% RSLogix 500 project LAB 5_BGJ.RSS, saved by version 8.40.00.08 %
PROJECT "MAN_MODE"    % processor: SLC 500, 1747-L541 %

PROGRAM FILES
  LAD 2   67 rungs

DATA FILES
  O0 OUTPUT  68 elements
  I1 INPUT  68 elements
  S2 STATUS  164 elements
  B3 BINARY  2 elements
  T4 TIMER  20 elements
  C5 COUNTER  2 elements
  R6 CONTROL  1 elements
  N7 INTEGER  1 elements
  F8 FLOAT  1 elements
  N10 PV_OUTPUTS  32 elements
  N11 PV_INPUTS  32 elements

LADDER 2
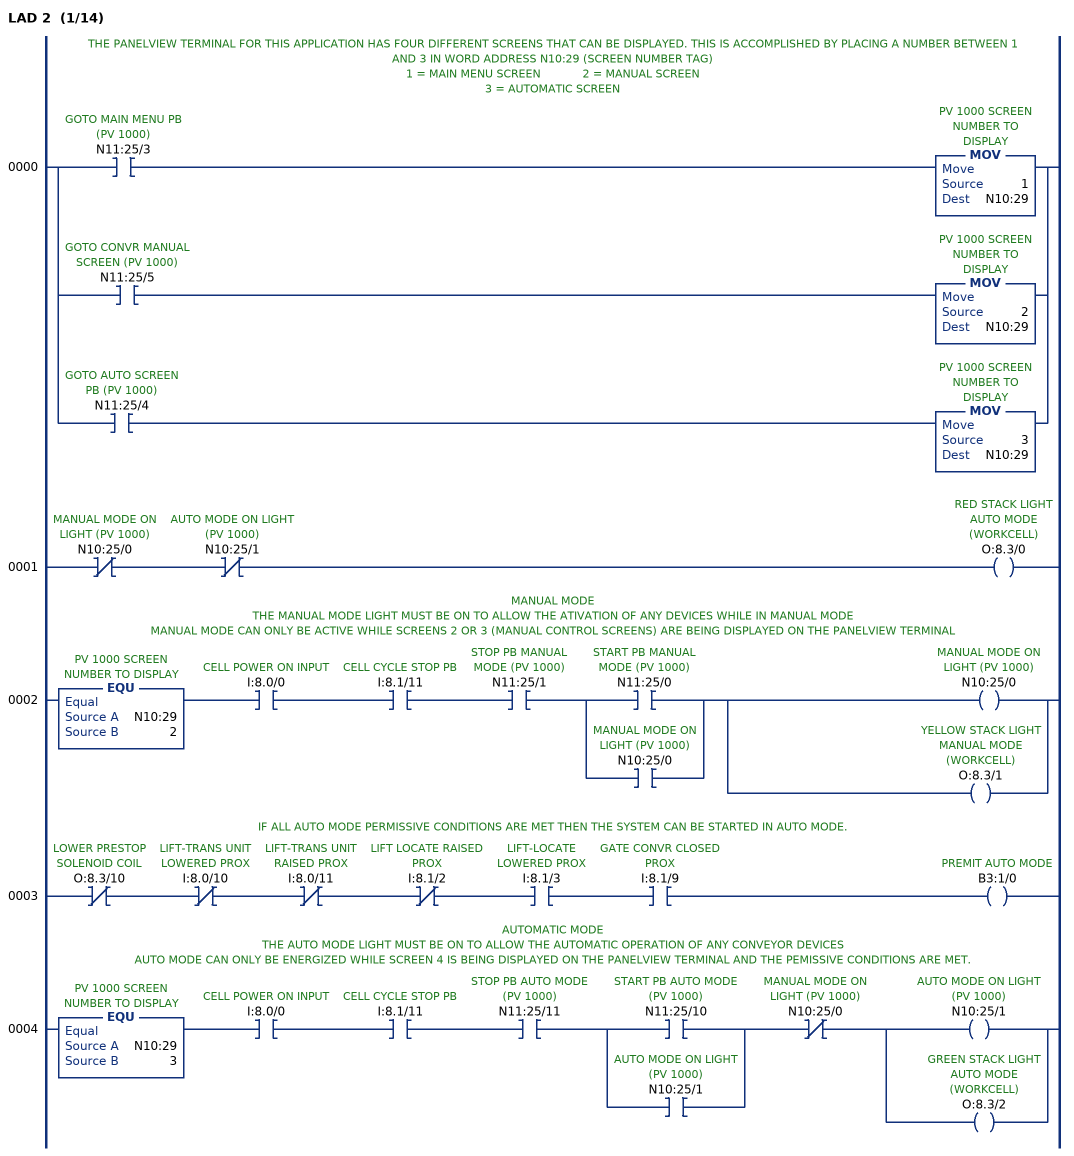
% Rung: 0 %
% THE PANELVIEW TERMINAL FOR THIS APPLICATION HAS FOUR DIFFERENT SCREENS THAT CAN BE DISPLAYED. THIS IS ACCOMPLISHED BY PLACING A NUMBER BETWEEN 1 AND 3 IN WORD ADDRESS N10:29 (SCREEN NUMBER TAG)
% 
% 1 = MAIN MENU SCREEN            2 = MANUAL SCREEN
% 3 = AUTOMATIC SCREEN %
SOR BST XIC N11:25/3 MOV 1 N10:29 NXB XIC N11:25/5 MOV 2 N10:29 NXB XIC N11:25/4 MOV 3 N10:29 BND EOR
%   N11:25/3  "GOTO MAIN MENU PB (PV 1000)" %
%   N10:29  "PV 1000 SCREEN NUMBER TO DISPLAY" %
%   N11:25/5  "GOTO CONVR MANUAL SCREEN (PV 1000)" %
%   N11:25/4  "GOTO AUTO SCREEN PB (PV 1000)" %
% Rung: 1 %
SOR XIO N10:25/0 XIO N10:25/1 OTE O:8.3/0 EOR
%   N10:25/0  "MANUAL MODE ON LIGHT (PV 1000)" %
%   N10:25/1  "AUTO MODE ON LIGHT (PV 1000)" %
%   O:8.3/0  "RED STACK LIGHT AUTO MODE (WORKCELL)" %
% Rung: 2 %
% MANUAL MODE
% 
% THE MANUAL MODE LIGHT MUST BE ON TO ALLOW THE ATIVATION OF ANY DEVICES WHILE IN MANUAL MODE
% MANUAL MODE CAN ONLY BE ACTIVE WHILE SCREENS 2 OR 3 (MANUAL CONTROL SCREENS) ARE BEING DISPLAYED ON THE PANELVIEW TERMINAL %
SOR EQU N10:29 2 XIC I:8.0/0 XIC I:8.1/11 XIC N11:25/1 BST XIC N11:25/0 NXB XIC N10:25/0 BND BST OTE N10:25/0 NXB OTE O:8.3/1 BND EOR
%   N10:29  "PV 1000 SCREEN NUMBER TO DISPLAY" %
%   I:8.0/0  "CELL POWER ON INPUT" %
%   I:8.1/11  "CELL CYCLE STOP PB" %
%   N11:25/1  "STOP PB MANUAL MODE (PV 1000)" %
%   N11:25/0  "START PB MANUAL MODE (PV 1000)" %
%   N10:25/0  "MANUAL MODE ON LIGHT (PV 1000)" %
%   O:8.3/1  "YELLOW STACK LIGHT MANUAL MODE (WORKCELL)" %
% Rung: 3 %
% IF ALL AUTO MODE PERMISSIVE CONDITIONS ARE MET THEN THE SYSTEM CAN BE STARTED IN AUTO MODE. %
SOR XIO O:8.3/10 XIO I:8.0/10 XIO I:8.0/11 XIO I:8.1/2 XIC I:8.1/3 XIC I:8.1/9 OTE B3:1/0 EOR
%   O:8.3/10  "LOWER PRESTOP SOLENOID COIL" %
%   I:8.0/10  "LIFT-TRANS UNIT LOWERED PROX" %
%   I:8.0/11  "LIFT-TRANS UNIT RAISED PROX" %
%   I:8.1/2  "LIFT LOCATE RAISED PROX" %
%   I:8.1/3  "LIFT-LOCATE LOWERED PROX" %
%   I:8.1/9  "GATE CONVR CLOSED PROX" %
%   B3:1/0  "PREMIT AUTO MODE" %
% Rung: 4 %
% AUTOMATIC MODE
% 
% THE AUTO MODE LIGHT MUST BE ON TO ALLOW THE AUTOMATIC OPERATION OF ANY CONVEYOR DEVICES
% 
% AUTO MODE CAN ONLY BE ENERGIZED WHILE SCREEN 4 IS BEING DISPLAYED ON THE PANELVIEW TERMINAL AND THE PEMISSIVE CONDITIONS ARE MET. %
SOR EQU N10:29 3 XIC I:8.0/0 XIC I:8.1/11 XIC N11:25/11 BST XIC N11:25/10 NXB XIC N10:25/1 BND XIO N10:25/0 BST OTE N10:25/1 NXB OTE O:8.3/2 BND EOR
%   N10:29  "PV 1000 SCREEN NUMBER TO DISPLAY" %
%   I:8.0/0  "CELL POWER ON INPUT" %
%   I:8.1/11  "CELL CYCLE STOP PB" %
%   N11:25/11  "STOP PB AUTO MODE (PV 1000)" %
%   N11:25/10  "START PB AUTO MODE (PV 1000)" %
%   N10:25/1  "AUTO MODE ON LIGHT (PV 1000)" %
%   N10:25/0  "MANUAL MODE ON LIGHT (PV 1000)" %
%   O:8.3/2  "GREEN STACK LIGHT AUTO MODE (WORKCELL)" %

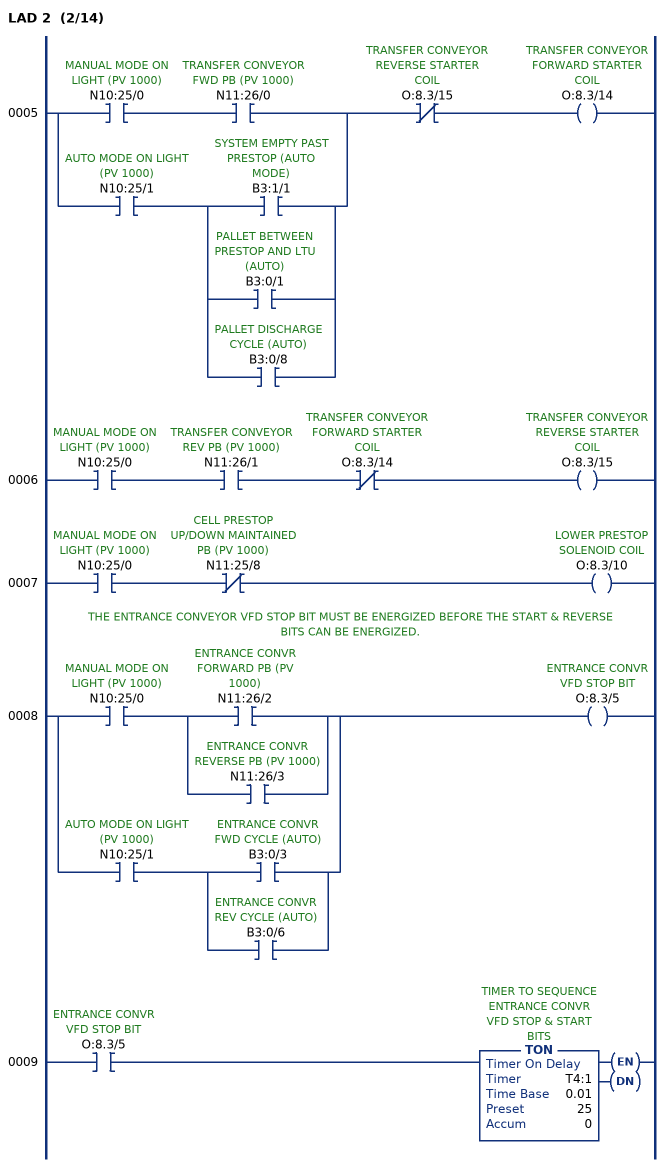
% Rung: 5 %
SOR BST XIC N10:25/0 XIC N11:26/0 NXB XIC N10:25/1 BST XIC B3:1/1 NXB XIC B3:0/1 NXB XIC B3:0/8 BND BND XIO O:8.3/15 OTE O:8.3/14 EOR
%   N10:25/0  "MANUAL MODE ON LIGHT (PV 1000)" %
%   N11:26/0  "TRANSFER CONVEYOR FWD PB (PV 1000)" %
%   N10:25/1  "AUTO MODE ON LIGHT (PV 1000)" %
%   B3:1/1  "SYSTEM EMPTY PAST PRESTOP (AUTO MODE)" %
%   B3:0/1  "PALLET BETWEEN PRESTOP AND LTU (AUTO)" %
%   B3:0/8  "PALLET DISCHARGE CYCLE (AUTO)" %
%   O:8.3/15  "TRANSFER CONVEYOR REVERSE STARTER COIL" %
%   O:8.3/14  "TRANSFER CONVEYOR FORWARD STARTER COIL" %
% Rung: 6 %
SOR XIC N10:25/0 XIC N11:26/1 XIO O:8.3/14 OTE O:8.3/15 EOR
%   N10:25/0  "MANUAL MODE ON LIGHT (PV 1000)" %
%   N11:26/1  "TRANSFER CONVEYOR REV PB (PV 1000)" %
%   O:8.3/14  "TRANSFER CONVEYOR FORWARD STARTER COIL" %
%   O:8.3/15  "TRANSFER CONVEYOR REVERSE STARTER COIL" %
% Rung: 7 %
SOR XIC N10:25/0 XIO N11:25/8 OTE O:8.3/10 EOR
%   N10:25/0  "MANUAL MODE ON LIGHT (PV 1000)" %
%   N11:25/8  "CELL PRESTOP UP/DOWN MAINTAINED PB (PV 1000)" %
%   O:8.3/10  "LOWER PRESTOP SOLENOID COIL" %
% Rung: 8 %
% THE ENTRANCE CONVEYOR VFD STOP BIT MUST BE ENERGIZED BEFORE THE START & REVERSE BITS CAN BE ENERGIZED. %
SOR BST XIC N10:25/0 BST XIC N11:26/2 NXB XIC N11:26/3 BND NXB XIC N10:25/1 BST XIC B3:0/3 NXB XIC B3:0/6 BND BND OTE O:8.3/5 EOR
%   N10:25/0  "MANUAL MODE ON LIGHT (PV 1000)" %
%   N11:26/2  "ENTRANCE CONVR FORWARD PB (PV 1000)" %
%   N11:26/3  "ENTRANCE CONVR REVERSE PB (PV 1000)" %
%   N10:25/1  "AUTO MODE ON LIGHT (PV 1000)" %
%   B3:0/3  "ENTRANCE CONVR FWD CYCLE (AUTO)" %
%   B3:0/6  "ENTRANCE CONVR REV CYCLE (AUTO)" %
%   O:8.3/5  "ENTRANCE CONVR VFD STOP BIT" %
% Rung: 9 %
SOR XIC O:8.3/5 TON T4:1 0.01 25 0 EOR
%   O:8.3/5  "ENTRANCE CONVR VFD STOP BIT" %
%   T4:1  "TIMER TO SEQUENCE ENTRANCE CONVR VFD STOP & START BITS" %

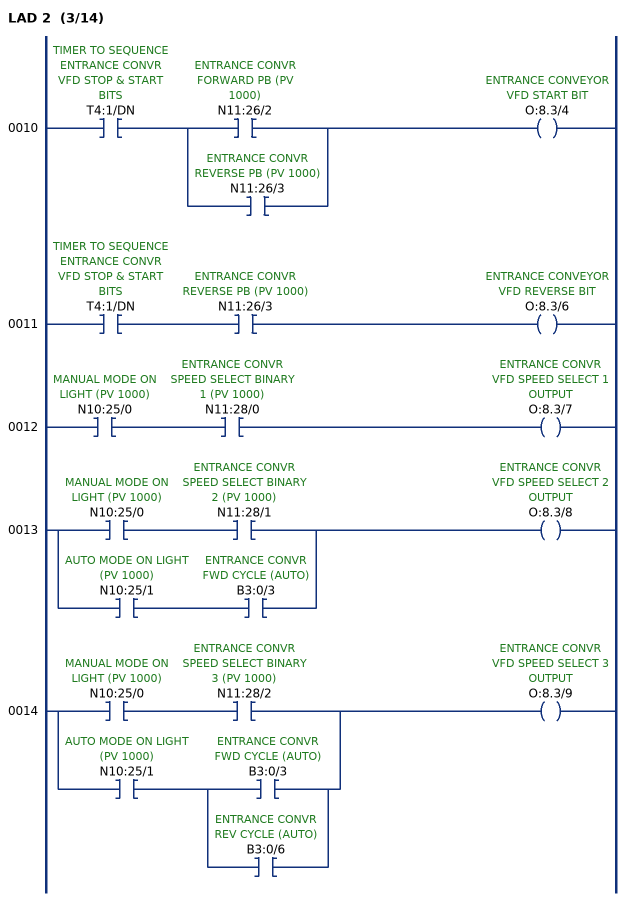
% Rung: 10 %
SOR XIC T4:1/DN BST XIC N11:26/2 NXB XIC N11:26/3 BND OTE O:8.3/4 EOR
%   T4:1  "TIMER TO SEQUENCE ENTRANCE CONVR VFD STOP & START BITS" %
%   N11:26/2  "ENTRANCE CONVR FORWARD PB (PV 1000)" %
%   N11:26/3  "ENTRANCE CONVR REVERSE PB (PV 1000)" %
%   O:8.3/4  "ENTRANCE CONVEYOR VFD START BIT" %
% Rung: 11 %
SOR XIC T4:1/DN XIC N11:26/3 OTE O:8.3/6 EOR
%   T4:1  "TIMER TO SEQUENCE ENTRANCE CONVR VFD STOP & START BITS" %
%   N11:26/3  "ENTRANCE CONVR REVERSE PB (PV 1000)" %
%   O:8.3/6  "ENTRANCE CONVEYOR VFD REVERSE BIT" %
% Rung: 12 %
SOR XIC N10:25/0 XIC N11:28/0 OTE O:8.3/7 EOR
%   N10:25/0  "MANUAL MODE ON LIGHT (PV 1000)" %
%   N11:28/0  "ENTRANCE CONVR SPEED SELECT BINARY 1 (PV 1000)" %
%   O:8.3/7  "ENTRANCE CONVR VFD SPEED SELECT 1 OUTPUT" %
% Rung: 13 %
SOR BST XIC N10:25/0 XIC N11:28/1 NXB XIC N10:25/1 XIC B3:0/3 BND OTE O:8.3/8 EOR
%   N10:25/0  "MANUAL MODE ON LIGHT (PV 1000)" %
%   N11:28/1  "ENTRANCE CONVR SPEED SELECT BINARY 2 (PV 1000)" %
%   N10:25/1  "AUTO MODE ON LIGHT (PV 1000)" %
%   B3:0/3  "ENTRANCE CONVR FWD CYCLE (AUTO)" %
%   O:8.3/8  "ENTRANCE CONVR VFD SPEED SELECT 2 OUTPUT" %
% Rung: 14 %
SOR BST XIC N10:25/0 XIC N11:28/2 NXB XIC N10:25/1 BST XIC B3:0/3 NXB XIC B3:0/6 BND BND OTE O:8.3/9 EOR
%   N10:25/0  "MANUAL MODE ON LIGHT (PV 1000)" %
%   N11:28/2  "ENTRANCE CONVR SPEED SELECT BINARY 3 (PV 1000)" %
%   N10:25/1  "AUTO MODE ON LIGHT (PV 1000)" %
%   B3:0/3  "ENTRANCE CONVR FWD CYCLE (AUTO)" %
%   B3:0/6  "ENTRANCE CONVR REV CYCLE (AUTO)" %
%   O:8.3/9  "ENTRANCE CONVR VFD SPEED SELECT 3 OUTPUT" %

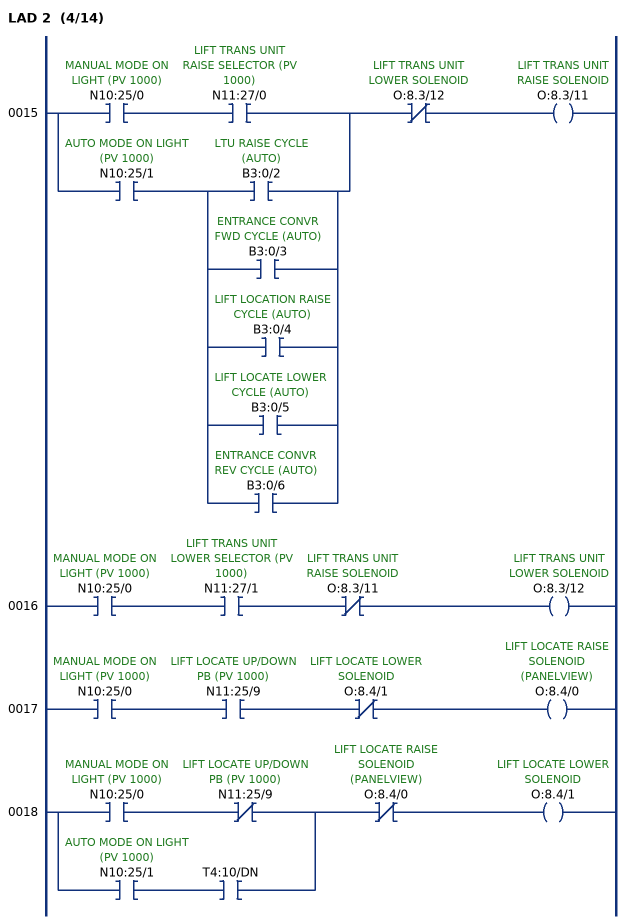
% Rung: 15 %
SOR BST XIC N10:25/0 XIC N11:27/0 NXB XIC N10:25/1 BST XIC B3:0/2 NXB XIC B3:0/3 NXB XIC B3:0/4 NXB XIC B3:0/5 NXB XIC B3:0/6 BND BND XIO O:8.3/12 OTE O:8.3/11 EOR
%   N10:25/0  "MANUAL MODE ON LIGHT (PV 1000)" %
%   N11:27/0  "LIFT TRANS UNIT RAISE SELECTOR (PV 1000)" %
%   N10:25/1  "AUTO MODE ON LIGHT (PV 1000)" %
%   B3:0/2  "LTU RAISE CYCLE (AUTO)" %
%   B3:0/3  "ENTRANCE CONVR FWD CYCLE (AUTO)" %
%   B3:0/4  "LIFT LOCATION RAISE CYCLE (AUTO)" %
%   B3:0/5  "LIFT LOCATE LOWER CYCLE (AUTO)" %
%   B3:0/6  "ENTRANCE CONVR REV CYCLE (AUTO)" %
%   O:8.3/12  "LIFT TRANS UNIT LOWER SOLENOID" %
%   O:8.3/11  "LIFT TRANS UNIT RAISE SOLENOID" %
% Rung: 16 %
SOR XIC N10:25/0 XIC N11:27/1 XIO O:8.3/11 OTE O:8.3/12 EOR
%   N10:25/0  "MANUAL MODE ON LIGHT (PV 1000)" %
%   N11:27/1  "LIFT TRANS UNIT LOWER SELECTOR (PV 1000)" %
%   O:8.3/11  "LIFT TRANS UNIT RAISE SOLENOID" %
%   O:8.3/12  "LIFT TRANS UNIT LOWER SOLENOID" %
% Rung: 17 %
SOR XIC N10:25/0 XIC N11:25/9 XIO O:8.4/1 OTE O:8.4/0 EOR
%   N10:25/0  "MANUAL MODE ON LIGHT (PV 1000)" %
%   N11:25/9  "LIFT LOCATE UP/DOWN PB (PV 1000)" %
%   O:8.4/1  "LIFT LOCATE LOWER SOLENOID" %
%   O:8.4/0  "LIFT LOCATE RAISE SOLENOID (PANELVIEW)" %
% Rung: 18 %
SOR BST XIC N10:25/0 XIO N11:25/9 NXB XIC N10:25/1 XIC T4:10/DN BND XIO O:8.4/0 OTE O:8.4/1 EOR
%   N10:25/0  "MANUAL MODE ON LIGHT (PV 1000)" %
%   N11:25/9  "LIFT LOCATE UP/DOWN PB (PV 1000)" %
%   N10:25/1  "AUTO MODE ON LIGHT (PV 1000)" %
%   O:8.4/0  "LIFT LOCATE RAISE SOLENOID (PANELVIEW)" %
%   O:8.4/1  "LIFT LOCATE LOWER SOLENOID" %

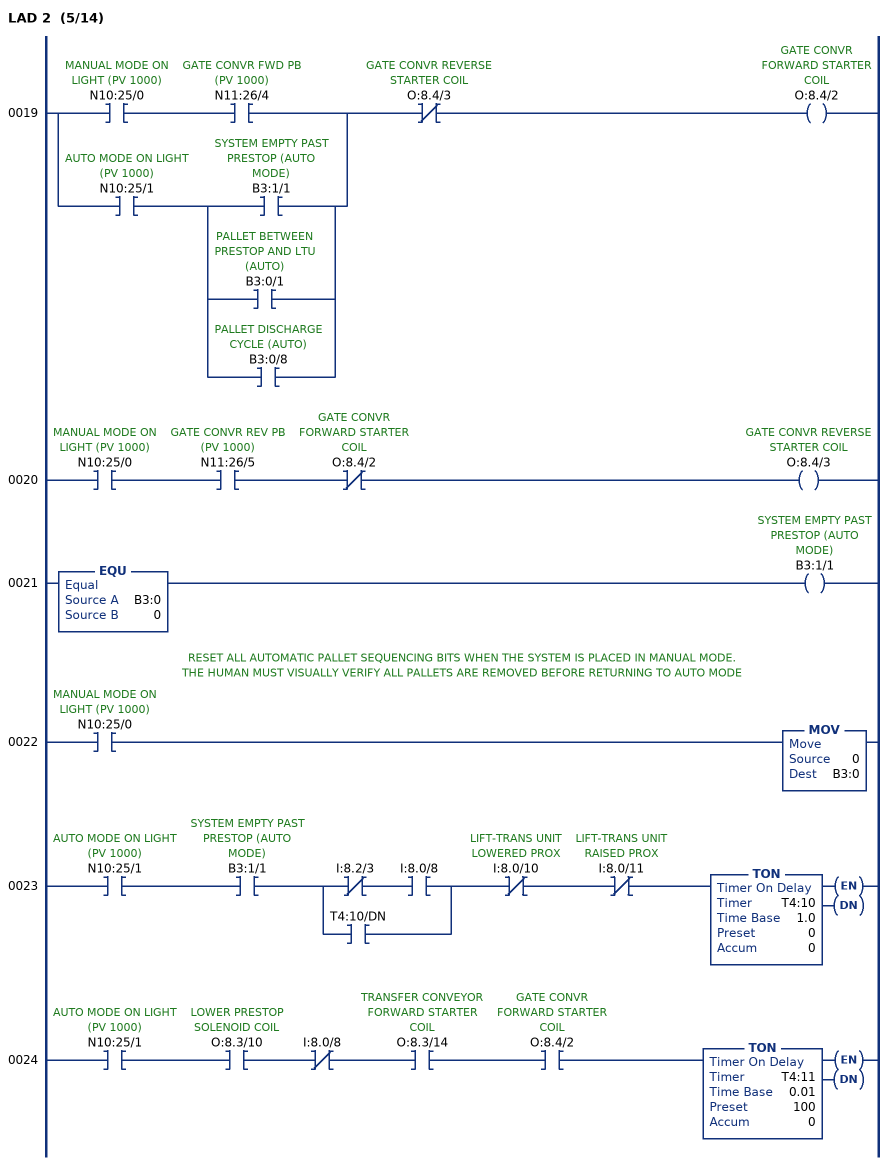
% Rung: 19 %
SOR BST XIC N10:25/0 XIC N11:26/4 NXB XIC N10:25/1 BST XIC B3:1/1 NXB XIC B3:0/1 NXB XIC B3:0/8 BND BND XIO O:8.4/3 OTE O:8.4/2 EOR
%   N10:25/0  "MANUAL MODE ON LIGHT (PV 1000)" %
%   N11:26/4  "GATE CONVR FWD PB (PV 1000)" %
%   N10:25/1  "AUTO MODE ON LIGHT (PV 1000)" %
%   B3:1/1  "SYSTEM EMPTY PAST PRESTOP (AUTO MODE)" %
%   B3:0/1  "PALLET BETWEEN PRESTOP AND LTU (AUTO)" %
%   B3:0/8  "PALLET DISCHARGE CYCLE (AUTO)" %
%   O:8.4/3  "GATE CONVR REVERSE STARTER COIL" %
%   O:8.4/2  "GATE CONVR FORWARD STARTER COIL" %
% Rung: 20 %
SOR XIC N10:25/0 XIC N11:26/5 XIO O:8.4/2 OTE O:8.4/3 EOR
%   N10:25/0  "MANUAL MODE ON LIGHT (PV 1000)" %
%   N11:26/5  "GATE CONVR REV PB (PV 1000)" %
%   O:8.4/2  "GATE CONVR FORWARD STARTER COIL" %
%   O:8.4/3  "GATE CONVR REVERSE STARTER COIL" %
% Rung: 21 %
SOR EQU B3:0 0 OTE B3:1/1 EOR
%   B3:1/1  "SYSTEM EMPTY PAST PRESTOP (AUTO MODE)" %
% Rung: 22 %
% RESET ALL AUTOMATIC PALLET SEQUENCING BITS WHEN THE SYSTEM IS PLACED IN MANUAL MODE.
% THE HUMAN MUST VISUALLY VERIFY ALL PALLETS ARE REMOVED BEFORE RETURNING TO AUTO MODE %
SOR XIC N10:25/0 MOV 0 B3:0 EOR
%   N10:25/0  "MANUAL MODE ON LIGHT (PV 1000)" %
% Rung: 23 %  % edit flag set %
SOR XIC N10:25/1 XIC B3:1/1 BST XIO I:8.2/3 XIC I:8.0/8 NXB XIC T4:10/DN BND XIO I:8.0/10 XIO I:8.0/11 TON T4:10 1.0 0 0 EOR
%   N10:25/1  "AUTO MODE ON LIGHT (PV 1000)" %
%   B3:1/1  "SYSTEM EMPTY PAST PRESTOP (AUTO MODE)" %
%   I:8.0/10  "LIFT-TRANS UNIT LOWERED PROX" %
%   I:8.0/11  "LIFT-TRANS UNIT RAISED PROX" %
% Rung: 24 %  % edit flag set %
SOR XIC N10:25/1 XIC O:8.3/10 XIO I:8.0/8 XIC O:8.3/14 XIC O:8.4/2 TON T4:11 0.01 100 0 EOR
%   N10:25/1  "AUTO MODE ON LIGHT (PV 1000)" %
%   O:8.3/10  "LOWER PRESTOP SOLENOID COIL" %
%   O:8.3/14  "TRANSFER CONVEYOR FORWARD STARTER COIL" %
%   O:8.4/2  "GATE CONVR FORWARD STARTER COIL" %

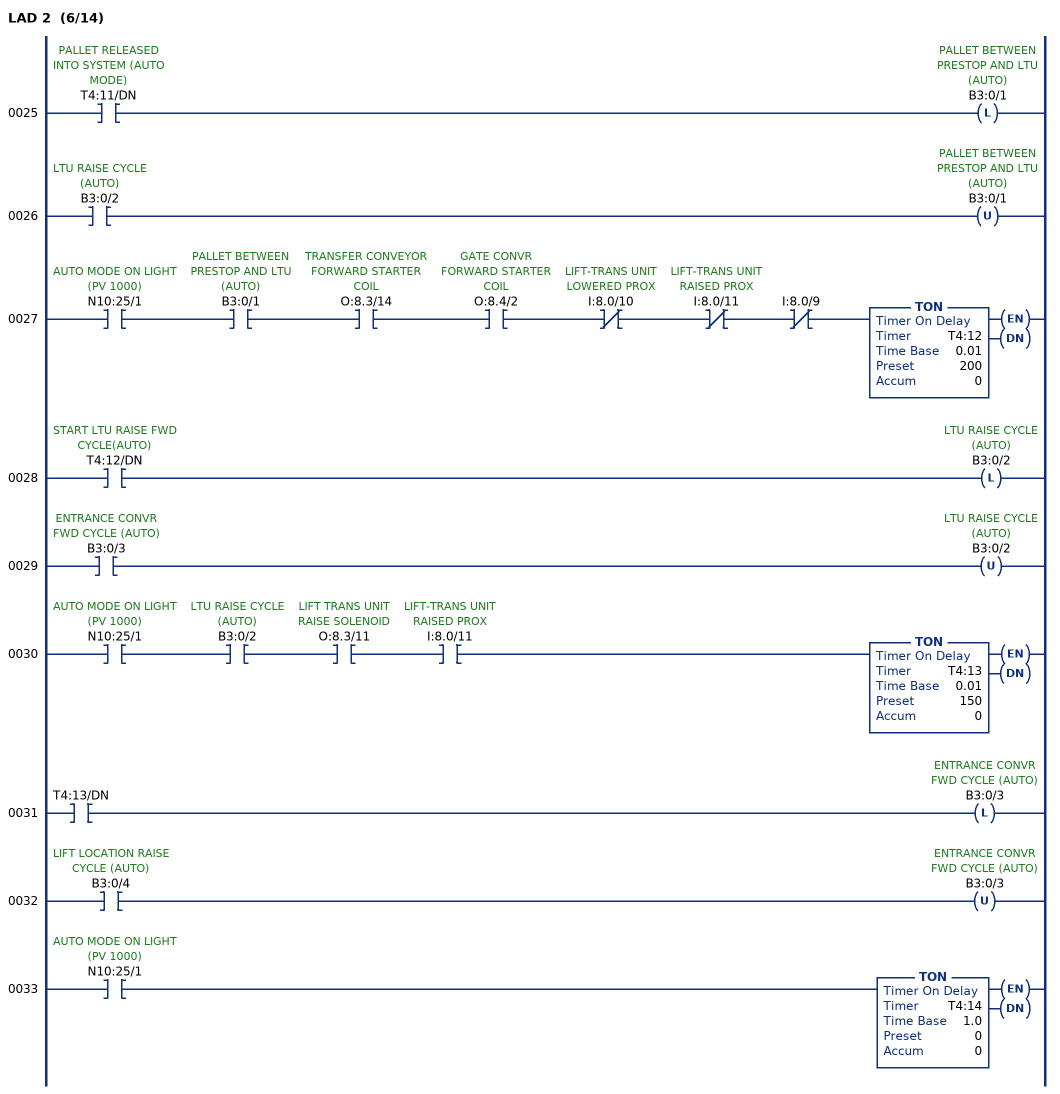
% Rung: 25 %  % edit flag set %
SOR XIC T4:11/DN OTL B3:0/1 EOR
%   T4:11/DN  "PALLET RELEASED INTO SYSTEM (AUTO MODE)" %
%   B3:0/1  "PALLET BETWEEN PRESTOP AND LTU (AUTO)" %
% Rung: 26 %  % edit flag set %
SOR XIC B3:0/2 OTU B3:0/1 EOR
%   B3:0/2  "LTU RAISE CYCLE (AUTO)" %
%   B3:0/1  "PALLET BETWEEN PRESTOP AND LTU (AUTO)" %
% Rung: 27 %  % edit flag set %
SOR XIC N10:25/1 XIC B3:0/1 XIC O:8.3/14 XIC O:8.4/2 XIO I:8.0/10 XIO I:8.0/11 XIO I:8.0/9 TON T4:12 0.01 200 0 EOR
%   N10:25/1  "AUTO MODE ON LIGHT (PV 1000)" %
%   B3:0/1  "PALLET BETWEEN PRESTOP AND LTU (AUTO)" %
%   O:8.3/14  "TRANSFER CONVEYOR FORWARD STARTER COIL" %
%   O:8.4/2  "GATE CONVR FORWARD STARTER COIL" %
%   I:8.0/10  "LIFT-TRANS UNIT LOWERED PROX" %
%   I:8.0/11  "LIFT-TRANS UNIT RAISED PROX" %
% Rung: 28 %  % edit flag set %
SOR XIC T4:12/DN OTL B3:0/2 EOR
%   T4:12/DN  "START LTU RAISE FWD CYCLE(AUTO)" %
%   B3:0/2  "LTU RAISE CYCLE (AUTO)" %
% Rung: 29 %  % edit flag set %
SOR XIC B3:0/3 OTU B3:0/2 EOR
%   B3:0/3  "ENTRANCE CONVR FWD CYCLE (AUTO)" %
%   B3:0/2  "LTU RAISE CYCLE (AUTO)" %
% Rung: 30 %  % edit flag set %
SOR XIC N10:25/1 XIC B3:0/2 XIC O:8.3/11 XIC I:8.0/11 TON T4:13 0.01 150 0 EOR
%   N10:25/1  "AUTO MODE ON LIGHT (PV 1000)" %
%   B3:0/2  "LTU RAISE CYCLE (AUTO)" %
%   O:8.3/11  "LIFT TRANS UNIT RAISE SOLENOID" %
%   I:8.0/11  "LIFT-TRANS UNIT RAISED PROX" %
% Rung: 31 %  % edit flag set %
SOR XIC T4:13/DN OTL B3:0/3 EOR
%   B3:0/3  "ENTRANCE CONVR FWD CYCLE (AUTO)" %
% Rung: 32 %  % edit flag set %
SOR XIC B3:0/4 OTU B3:0/3 EOR
%   B3:0/4  "LIFT LOCATION RAISE CYCLE (AUTO)" %
%   B3:0/3  "ENTRANCE CONVR FWD CYCLE (AUTO)" %
% Rung: 33 %  % edit flag set %
SOR XIC N10:25/1 TON T4:14 1.0 0 0 EOR
%   N10:25/1  "AUTO MODE ON LIGHT (PV 1000)" %

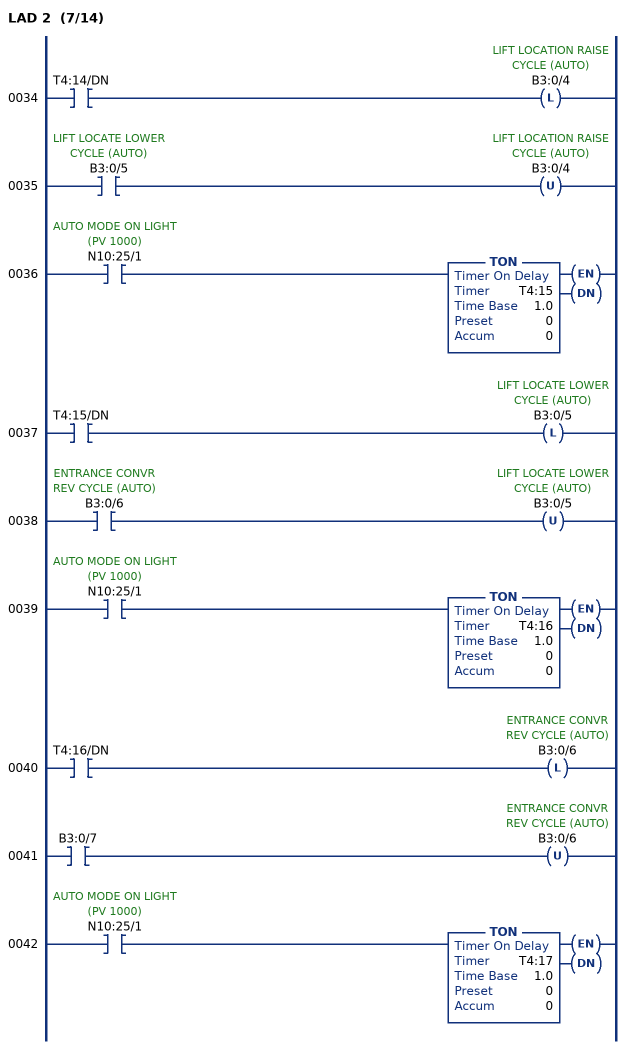
% Rung: 34 %  % edit flag set %
SOR XIC T4:14/DN OTL B3:0/4 EOR
%   B3:0/4  "LIFT LOCATION RAISE CYCLE (AUTO)" %
% Rung: 35 %  % edit flag set %
SOR XIC B3:0/5 OTU B3:0/4 EOR
%   B3:0/5  "LIFT LOCATE LOWER CYCLE (AUTO)" %
%   B3:0/4  "LIFT LOCATION RAISE CYCLE (AUTO)" %
% Rung: 36 %  % edit flag set %
SOR XIC N10:25/1 TON T4:15 1.0 0 0 EOR
%   N10:25/1  "AUTO MODE ON LIGHT (PV 1000)" %
% Rung: 37 %  % edit flag set %
SOR XIC T4:15/DN OTL B3:0/5 EOR
%   B3:0/5  "LIFT LOCATE LOWER CYCLE (AUTO)" %
% Rung: 38 %  % edit flag set %
SOR XIC B3:0/6 OTU B3:0/5 EOR
%   B3:0/6  "ENTRANCE CONVR REV CYCLE (AUTO)" %
%   B3:0/5  "LIFT LOCATE LOWER CYCLE (AUTO)" %
% Rung: 39 %  % edit flag set %
SOR XIC N10:25/1 TON T4:16 1.0 0 0 EOR
%   N10:25/1  "AUTO MODE ON LIGHT (PV 1000)" %
% Rung: 40 %  % edit flag set %
SOR XIC T4:16/DN OTL B3:0/6 EOR
%   B3:0/6  "ENTRANCE CONVR REV CYCLE (AUTO)" %
% Rung: 41 %  % edit flag set %
SOR XIC B3:0/7 OTU B3:0/6 EOR
%   B3:0/6  "ENTRANCE CONVR REV CYCLE (AUTO)" %
% Rung: 42 %  % edit flag set %
SOR XIC N10:25/1 TON T4:17 1.0 0 0 EOR
%   N10:25/1  "AUTO MODE ON LIGHT (PV 1000)" %

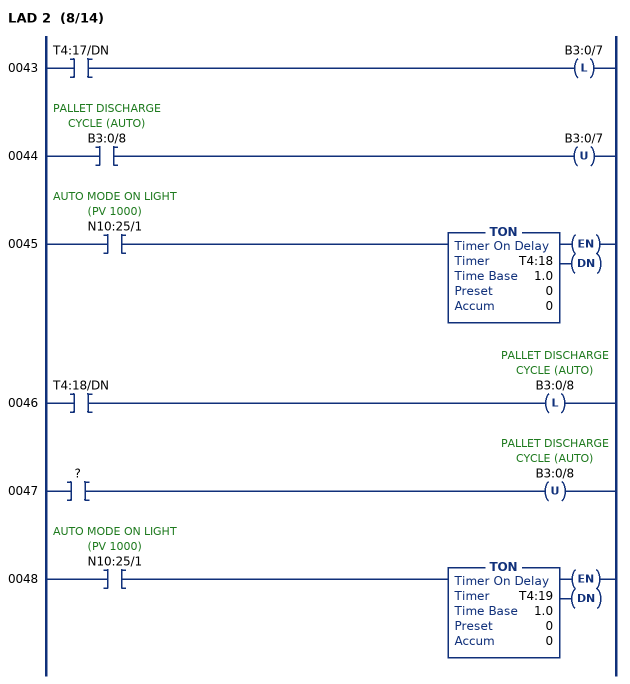
% Rung: 43 %  % edit flag set %
SOR XIC T4:17/DN OTL B3:0/7 EOR
% Rung: 44 %  % edit flag set %
SOR XIC B3:0/8 OTU B3:0/7 EOR
%   B3:0/8  "PALLET DISCHARGE CYCLE (AUTO)" %
% Rung: 45 %  % edit flag set %
SOR XIC N10:25/1 TON T4:18 1.0 0 0 EOR
%   N10:25/1  "AUTO MODE ON LIGHT (PV 1000)" %
% Rung: 46 %  % edit flag set %
SOR XIC T4:18/DN OTL B3:0/8 EOR
%   B3:0/8  "PALLET DISCHARGE CYCLE (AUTO)" %
% Rung: 47 %  % edit flag set %
SOR XIC ? OTU B3:0/8 EOR
%   B3:0/8  "PALLET DISCHARGE CYCLE (AUTO)" %
% Rung: 48 %  % edit flag set %
SOR XIC N10:25/1 TON T4:19 1.0 0 0 EOR
%   N10:25/1  "AUTO MODE ON LIGHT (PV 1000)" %

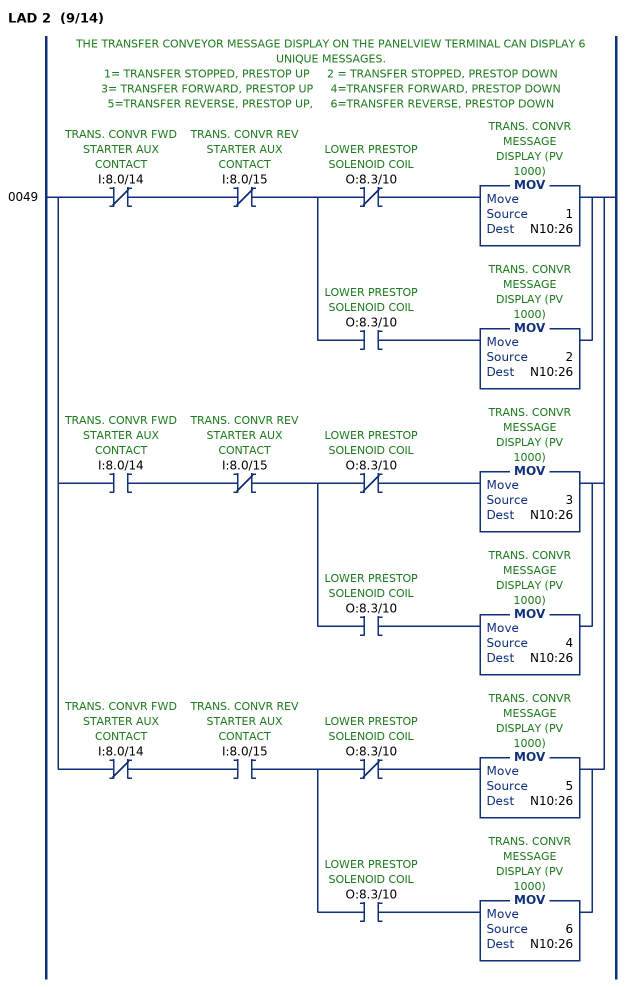
% Rung: 49 %
% THE TRANSFER CONVEYOR MESSAGE DISPLAY ON THE PANELVIEW TERMINAL CAN DISPLAY 6 UNIQUE MESSAGES.
% 1= TRANSFER STOPPED, PRESTOP UP     2 = TRANSFER STOPPED, PRESTOP DOWN
% 3= TRANSFER FORWARD, PRESTOP UP     4=TRANSFER FORWARD, PRESTOP DOWN
% 5=TRANSFER REVERSE, PRESTOP UP,     6=TRANSFER REVERSE, PRESTOP DOWN %
SOR BST XIO I:8.0/14 XIO I:8.0/15 BST XIO O:8.3/10 MOV 1 N10:26 NXB XIC O:8.3/10 MOV 2 N10:26 BND NXB XIC I:8.0/14 XIO I:8.0/15 BST XIO O:8.3/10 MOV 3 N10:26 NXB XIC O:8.3/10 MOV 4 N10:26 BND NXB XIO I:8.0/14 XIC I:8.0/15 BST XIO O:8.3/10 MOV 5 N10:26 NXB XIC O:8.3/10 MOV 6 N10:26 BND BND EOR
%   I:8.0/14  "TRANS. CONVR FWD STARTER AUX CONTACT" %
%   I:8.0/15  "TRANS. CONVR REV STARTER AUX CONTACT" %
%   O:8.3/10  "LOWER PRESTOP SOLENOID COIL" %
%   N10:26  "TRANS. CONVR MESSAGE DISPLAY (PV 1000)" %

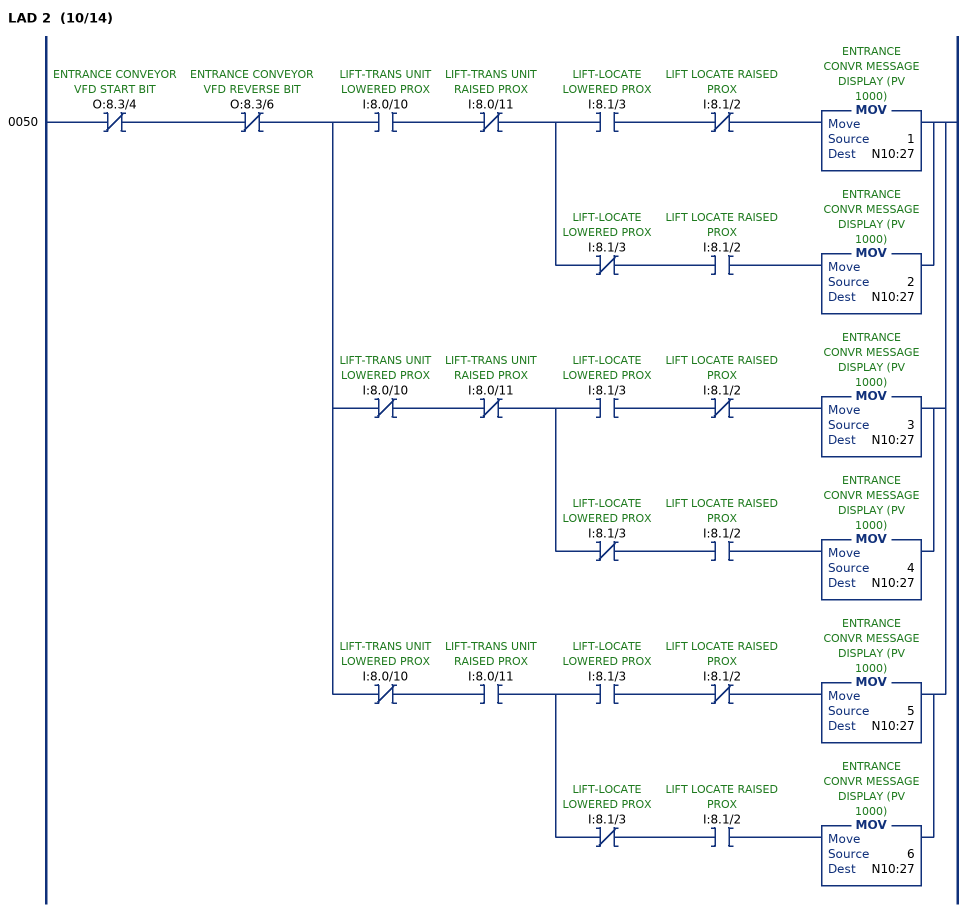
% Rung: 50 %
SOR XIO O:8.3/4 XIO O:8.3/6 BST XIC I:8.0/10 XIO I:8.0/11 BST XIC I:8.1/3 XIO I:8.1/2 MOV 1 N10:27 NXB XIO I:8.1/3 XIC I:8.1/2 MOV 2 N10:27 BND NXB XIO I:8.0/10 XIO I:8.0/11 BST XIC I:8.1/3 XIO I:8.1/2 MOV 3 N10:27 NXB XIO I:8.1/3 XIC I:8.1/2 MOV 4 N10:27 BND NXB XIO I:8.0/10 XIC I:8.0/11 BST XIC I:8.1/3 XIO I:8.1/2 MOV 5 N10:27 NXB XIO I:8.1/3 XIC I:8.1/2 MOV 6 N10:27 BND BND EOR
%   O:8.3/4  "ENTRANCE CONVEYOR VFD START BIT" %
%   O:8.3/6  "ENTRANCE CONVEYOR VFD REVERSE BIT" %
%   I:8.0/10  "LIFT-TRANS UNIT LOWERED PROX" %
%   I:8.0/11  "LIFT-TRANS UNIT RAISED PROX" %
%   I:8.1/3  "LIFT-LOCATE LOWERED PROX" %
%   I:8.1/2  "LIFT LOCATE RAISED PROX" %
%   N10:27  "ENTRANCE CONVR MESSAGE DISPLAY (PV 1000)" %

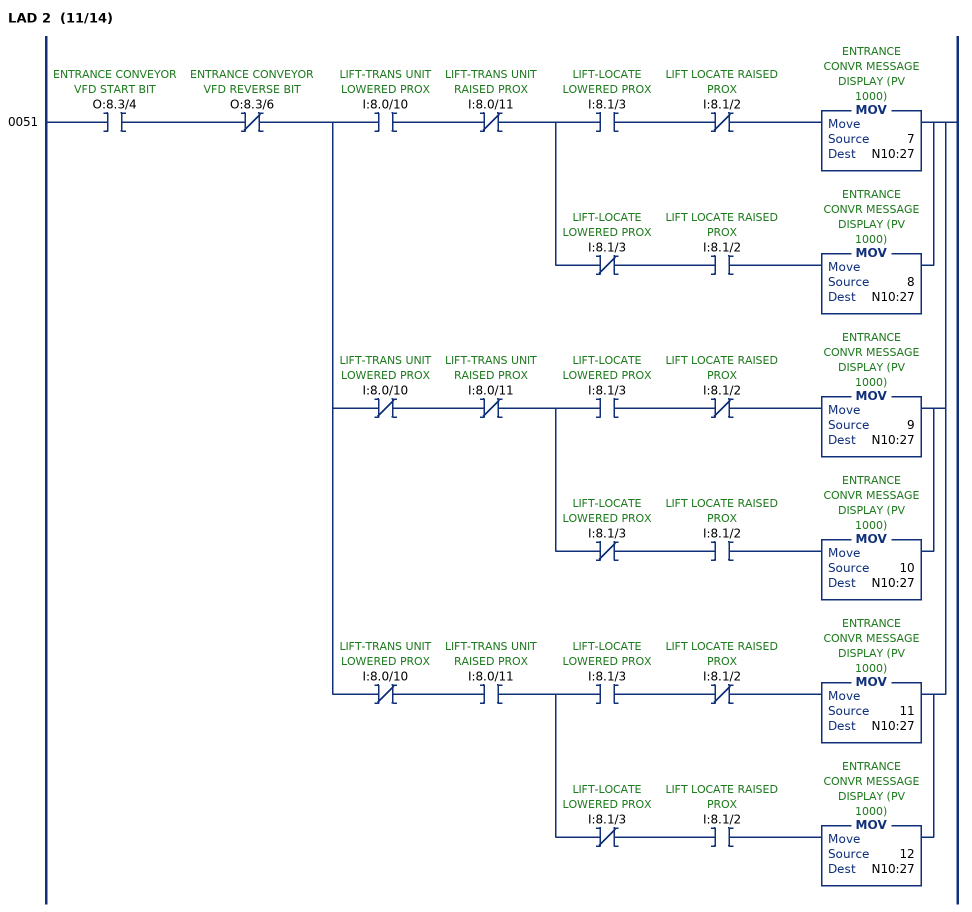
% Rung: 51 %
SOR XIC O:8.3/4 XIO O:8.3/6 BST XIC I:8.0/10 XIO I:8.0/11 BST XIC I:8.1/3 XIO I:8.1/2 MOV 7 N10:27 NXB XIO I:8.1/3 XIC I:8.1/2 MOV 8 N10:27 BND NXB XIO I:8.0/10 XIO I:8.0/11 BST XIC I:8.1/3 XIO I:8.1/2 MOV 9 N10:27 NXB XIO I:8.1/3 XIC I:8.1/2 MOV 10 N10:27 BND NXB XIO I:8.0/10 XIC I:8.0/11 BST XIC I:8.1/3 XIO I:8.1/2 MOV 11 N10:27 NXB XIO I:8.1/3 XIC I:8.1/2 MOV 12 N10:27 BND BND EOR
%   O:8.3/4  "ENTRANCE CONVEYOR VFD START BIT" %
%   O:8.3/6  "ENTRANCE CONVEYOR VFD REVERSE BIT" %
%   I:8.0/10  "LIFT-TRANS UNIT LOWERED PROX" %
%   I:8.0/11  "LIFT-TRANS UNIT RAISED PROX" %
%   I:8.1/3  "LIFT-LOCATE LOWERED PROX" %
%   I:8.1/2  "LIFT LOCATE RAISED PROX" %
%   N10:27  "ENTRANCE CONVR MESSAGE DISPLAY (PV 1000)" %

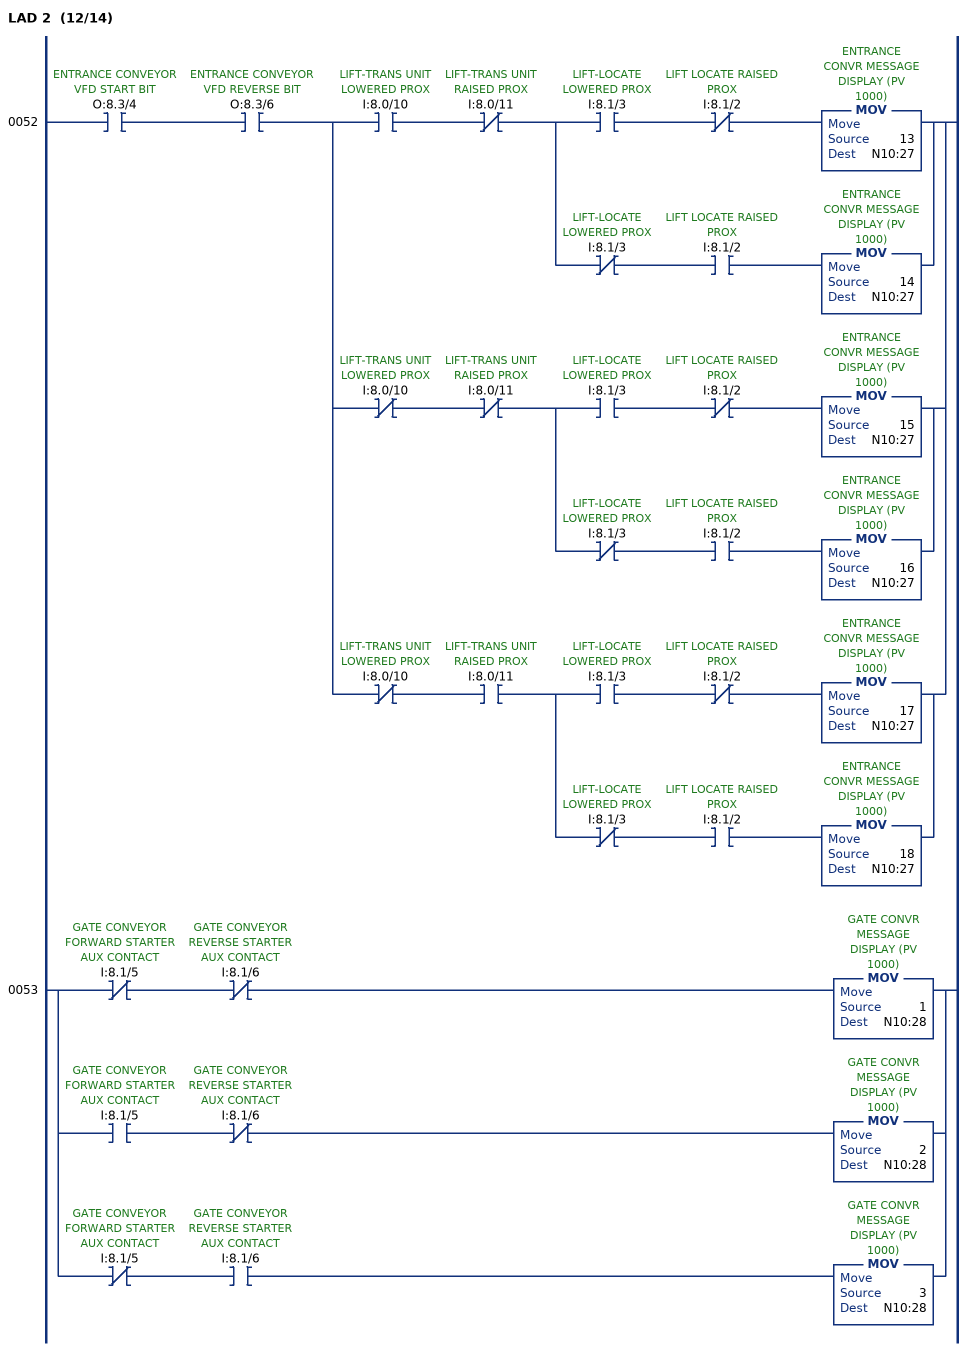
% Rung: 52 %
SOR XIC O:8.3/4 XIC O:8.3/6 BST XIC I:8.0/10 XIO I:8.0/11 BST XIC I:8.1/3 XIO I:8.1/2 MOV 13 N10:27 NXB XIO I:8.1/3 XIC I:8.1/2 MOV 14 N10:27 BND NXB XIO I:8.0/10 XIO I:8.0/11 BST XIC I:8.1/3 XIO I:8.1/2 MOV 15 N10:27 NXB XIO I:8.1/3 XIC I:8.1/2 MOV 16 N10:27 BND NXB XIO I:8.0/10 XIC I:8.0/11 BST XIC I:8.1/3 XIO I:8.1/2 MOV 17 N10:27 NXB XIO I:8.1/3 XIC I:8.1/2 MOV 18 N10:27 BND BND EOR
%   O:8.3/4  "ENTRANCE CONVEYOR VFD START BIT" %
%   O:8.3/6  "ENTRANCE CONVEYOR VFD REVERSE BIT" %
%   I:8.0/10  "LIFT-TRANS UNIT LOWERED PROX" %
%   I:8.0/11  "LIFT-TRANS UNIT RAISED PROX" %
%   I:8.1/3  "LIFT-LOCATE LOWERED PROX" %
%   I:8.1/2  "LIFT LOCATE RAISED PROX" %
%   N10:27  "ENTRANCE CONVR MESSAGE DISPLAY (PV 1000)" %
% Rung: 53 %
SOR BST XIO I:8.1/5 XIO I:8.1/6 MOV 1 N10:28 NXB XIC I:8.1/5 XIO I:8.1/6 MOV 2 N10:28 NXB XIO I:8.1/5 XIC I:8.1/6 MOV 3 N10:28 BND EOR
%   I:8.1/5  "GATE CONVEYOR FORWARD STARTER AUX CONTACT" %
%   I:8.1/6  "GATE CONVEYOR REVERSE STARTER AUX CONTACT" %
%   N10:28  "GATE CONVR MESSAGE DISPLAY (PV 1000)" %

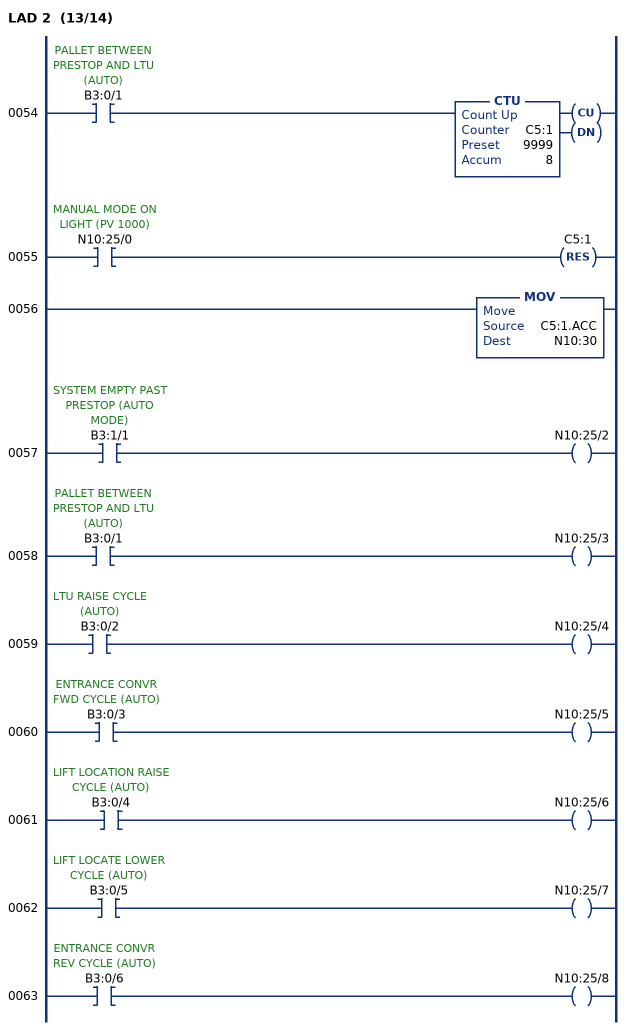
% Rung: 54 %  % edit flag set %
SOR XIC B3:0/1 CTU C5:1 9999 8 EOR
%   B3:0/1  "PALLET BETWEEN PRESTOP AND LTU (AUTO)" %
% Rung: 55 %  % edit flag set %
SOR XIC N10:25/0 RES C5:1 EOR
%   N10:25/0  "MANUAL MODE ON LIGHT (PV 1000)" %
% Rung: 56 %  % edit flag set %
SOR MOV C5:1.ACC N10:30 EOR
% Rung: 57 %  % edit flag set %
SOR XIC B3:1/1 OTE N10:25/2 EOR
%   B3:1/1  "SYSTEM EMPTY PAST PRESTOP (AUTO MODE)" %
% Rung: 58 %  % edit flag set %
SOR XIC B3:0/1 OTE N10:25/3 EOR
%   B3:0/1  "PALLET BETWEEN PRESTOP AND LTU (AUTO)" %
% Rung: 59 %  % edit flag set %
SOR XIC B3:0/2 OTE N10:25/4 EOR
%   B3:0/2  "LTU RAISE CYCLE (AUTO)" %
% Rung: 60 %  % edit flag set %
SOR XIC B3:0/3 OTE N10:25/5 EOR
%   B3:0/3  "ENTRANCE CONVR FWD CYCLE (AUTO)" %
% Rung: 61 %  % edit flag set %
SOR XIC B3:0/4 OTE N10:25/6 EOR
%   B3:0/4  "LIFT LOCATION RAISE CYCLE (AUTO)" %
% Rung: 62 %  % edit flag set %
SOR XIC B3:0/5 OTE N10:25/7 EOR
%   B3:0/5  "LIFT LOCATE LOWER CYCLE (AUTO)" %
% Rung: 63 %  % edit flag set %
SOR XIC B3:0/6 OTE N10:25/8 EOR
%   B3:0/6  "ENTRANCE CONVR REV CYCLE (AUTO)" %

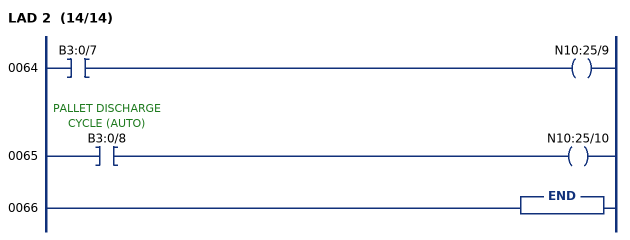
% Rung: 64 %  % edit flag set %
SOR XIC B3:0/7 OTE N10:25/9 EOR
% Rung: 65 %  % edit flag set %
SOR XIC B3:0/8 OTE N10:25/10 EOR
%   B3:0/8  "PALLET DISCHARGE CYCLE (AUTO)" %
% Rung: 66 %
SOR END EOR

OTHER DOCUMENTED ADDRESSES
  AUTO  "AUTO MODE LIGHT"

COMMENTS NOT ATTACHED TO A CURRENT RUNG
  O:2.0/8: 5LT - STEP 5
  O:2.0/0: A PAGE TITLE CAUSES THE PROGRAM PRINTOUT TO START AT A NEW PAGE / SYSTEM STOP 1PBLT - RUNG COMMENT
  O:2.0/1: 2PBLT GREEN BUTTON AND LIGHT - RUNG COMMENT
  O:2.0/2: STEP 2 - 3PBLT
  O:2.0/4: STEP 1
  B3:0/0: IF ALL CONDITIONS ON THIS RUNG ARE MET, THEN THE SYSTEM CAN BE STARTED IN AUTOMATIC MODE.
  O:2.0/10: STEP 3 - HORN
  O:2.0/9: 6LT - STEP 4
  O:8.29: THE PANELVIEW TERMINAL FOR THIS APPLICATION HAS FOUR DIFFERENT SCREENS THAT CAN BE DISPLAYED. THIS IS ACCOMPLISHED BY PLACING A NUMBER BETWEEN 1 AND 4 IN WORD ADDRESS O:8.29 (SCREEN NUMBER TAG)
    
    1 = MAIN MENU SCREEN            2 = MANUAL SCREEN_1
    3 = MANUAL SCREEN_2            4 AUTOMATIC SCREEN
  O:8.26: THE TRANSFER CONVEYOR MESSAGE DISPLAY ON THE PANELVIEW TERMINAL CAN DISPLAY 6 UNIQUE MESSAGES.
    1= TRANSFER STOPPED, PRESTOP UP     2 = TRANSFER STOPPED, PRESTOP DOWN
    3= TRANSFER FORWARD, PRESTOP UP     4=TRANSFER FORWARD, PRESTOP DOWN
    5=TRANSFER REVERSE, PRESTOP UP,     6=TRANSFER REVERSE, PRESTOP DOWN
  O:8.27: THE ENTRANCE CONVEYOR MESSAGE DISPLAY ON THE PANELVIEW TERMINAL CAN DISPLAY 18 UNIQUE MESSAGES.
    1= ENTRANCE STOPPED, LTU LOWERED, LIFT DOWN     2 = ENTRANCE STOPPED, LTU LOWERED, LIFT UP     3=ENTRANCE STOPPED, LTU CENTRED, LIFT DOWN
    4= ENTRANCE STOPPED, LTU CENTRED, LIFT UP     5 = ENTRANCE STOPPED, LTU RAISED, LIFT DOWN     6=ENTRANCE STOPPED, LTU RAISED, LIFT UP
    7= ENTRANCE FORWARD, LTU LOWERED, LIFT DOWN     8 = ENTRANCE FORWARD, LTU LOWERED, LIFT UP     9=ENTRANCE FORWARD, LTU CENTRED, LIFT DOWN
    10= ENTRANCE FORWARD, LTU CENTRED, LIFT UP     11 = ENTRANCE FORWARD, LTU RAISED, LIFT DOWN     12=ENTRANCE STOPPED, LTU RAISED, LIFT UP
    13= ENTRANCE REVERSE, LTU LOWERED, LIFT DOWN     14 = ENTRANCE REVERSE, LTU LOWERED, LIFT UP     15=ENTRANCE REVERSE, LTU CENTRED, LIFT DOWN
    16= ENTRANCE REVERSE, LTU CENTRED, LIFT UP     17 = ENTRANCE REVERSE, LTU RAISED, LIFT DOWN     18=ENTRANCE REVERSE, LTU RAISED, LIFT UP

DATA TABLE (non-zero values as saved)
DATA B3
% B3:0 % 0X0000 0X0003
DATA T4
% .PRE .ACC %
% T4:1 % 25 0
% T4:10 % 300 0
% T4:11 % 100 0
% T4:12 % 200 0
% T4:13 % 150 0
% T4:14 % 250 0
% T4:15 % 400 0
% T4:16 % 200 0
% T4:17 % 150 0
% T4:18 % 250 0
% T4:19 % 500 0
DATA C5
% .PRE .ACC %
% C5:1 % 9999 8
DATA N10
% N10:20 % 0 0 0 0 0 0 1 3 1 3
DATA N11
% N11:20 % 0 0 0 0 0 2050 0 2 5 0
